TYPE "udt_DeviceSafetyInterface"
VERSION : 0.1
// Block: udt_DeviceSafetyInterface
   STRUCT
      SafeStop : Bool;
      PowerEnable : Bool;
      DevicesInSafeState : Bool;
   END_STRUCT;

END_TYPE
